// LS Electric XG5000 project: 16-41-1
// PLC NewPLC
// module base 0 slot 0: 입출력 모듈:XBC-DR14E (DC 24V 입력 8점, 릴레이 출력 6점)

PROGRAM NewProgram (task: 스캔 프로그램)

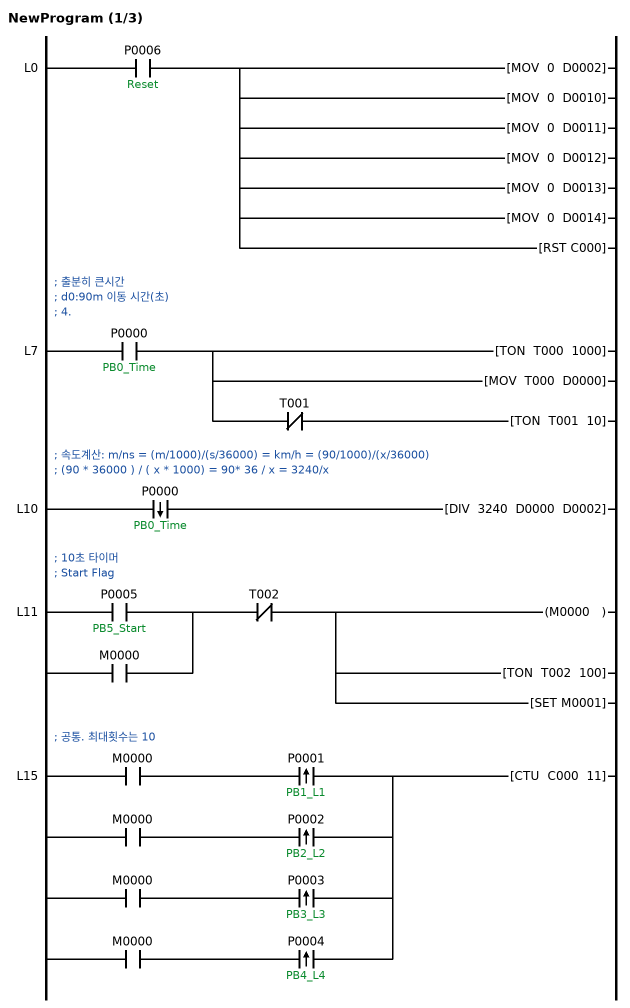
; L0
LOAD      P0006	// Reset
MOV       0 D0002
MOV       0 D0010
MOV       0 D0011
MOV       0 D0012
MOV       0 D0013
MOV       0 D0014
RST       C000
; L7
LOAD      P0000	// PB0_Time
TON       T000 1000
MOV       T000 D0000
AND NOT   T001
TON       T001 10
// output comment: 출분히 큰시간
// output comment: d0:90m 이동 시간(초)
// output comment: 4.
; L10
LOADN     P0000	// PB0_Time
DIV       3240 D0000 D0002
// output comment: 속도계산: m/ns = (m/1000)/(s/36000) = km/h = (90/1000)/(x/36000)           (90 * 36000 ) / ( x * 1000) = 90* 36 / x = 3240/x
; L11
LOAD      P0005	// PB5_Start
OR        M0000
AND NOT   T002
OUT       M0000
TON       T002 100
SET       M0001
// output comment: 10초 타이머
// output comment: Start Flag
; L15
LOAD      M0000
ANDP      P0001	// PB1_L1
LOAD      M0000
ANDP      P0002	// PB2_L2
OR LOAD
LOAD      M0000
ANDP      P0003	// PB3_L3
OR LOAD
LOAD      M0000
ANDP      P0004	// PB4_L4
OR LOAD
CTU       C000 11
// output comment: 공통. 최대횟수는 10

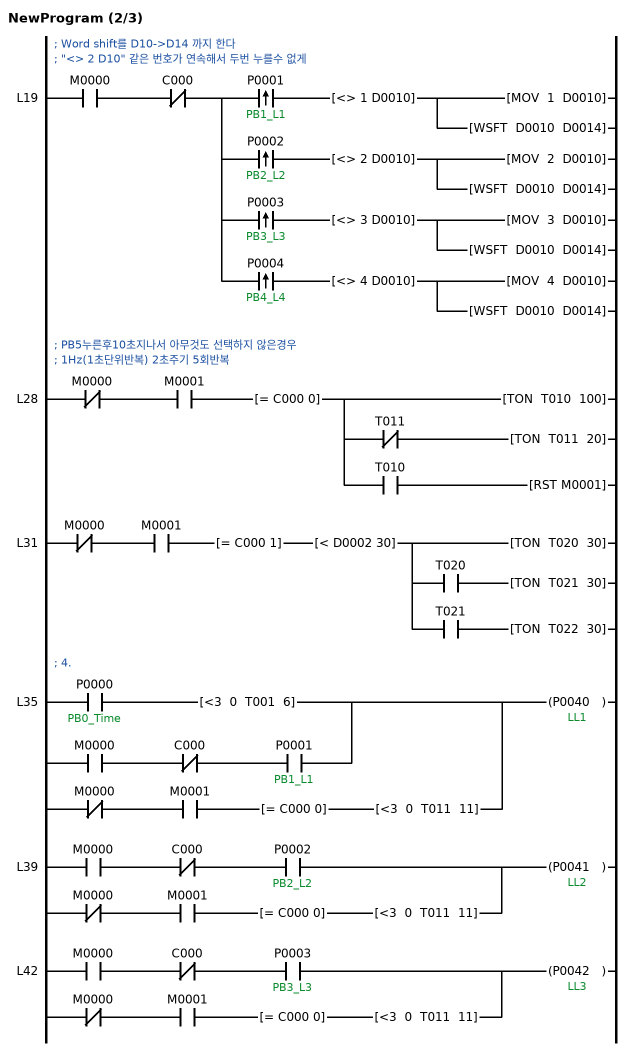
; L19
LOAD      M0000
AND NOT   C000
MPUSH
ANDP      P0001	// PB1_L1
AND<>     1 D0010
MOV       1 D0010
WSFT      D0010 D0014
MLOAD
ANDP      P0002	// PB2_L2
AND<>     2 D0010
MOV       2 D0010
WSFT      D0010 D0014
MLOAD
ANDP      P0003	// PB3_L3
AND<>     3 D0010
MOV       3 D0010
WSFT      D0010 D0014
MPOP
ANDP      P0004	// PB4_L4
AND<>     4 D0010
MOV       4 D0010
WSFT      D0010 D0014
// output comment: Word shift를 D10->D14 까지 한다
// output comment: "<> 2 D10" 같은 번호가 연속해서 두번 누를수 없게 
; L28
LOAD NOT  M0000
AND       M0001
AND=      C000 0
TON       T010 100
MPUSH
AND NOT   T011
TON       T011 20
MPOP
AND       T010
RST       M0001
// output comment: PB5누른후10초지나서 아무것도 선택하지 않은경우
// output comment: 1Hz(1초단위반복) 2초주기 5회반복
; L31
LOAD NOT  M0000
AND       M0001
AND=      C000 1
AND<      D0002 30
TON       T020 30
MPUSH
AND       T020
TON       T021 30
MPOP
AND       T021
TON       T022 30
; L35
LOAD      P0000	// PB0_Time
AND<3     0 T001 6
LOAD      M0000
AND NOT   C000
AND       P0001	// PB1_L1
OR LOAD
LOAD NOT  M0000
AND       M0001
AND=      C000 0
AND<3     0 T011 11
OR LOAD
OUT       P0040	// LL1
// output comment: 4.
; L39
LOAD      M0000
AND NOT   C000
AND       P0002	// PB2_L2
LOAD NOT  M0000
AND       M0001
AND=      C000 0
AND<3     0 T011 11
OR LOAD
OUT       P0041	// LL2
; L42
LOAD      M0000
AND NOT   C000
AND       P0003	// PB3_L3
LOAD NOT  M0000
AND       M0001
AND=      C000 0
AND<3     0 T011 11
OR LOAD
OUT       P0042	// LL3

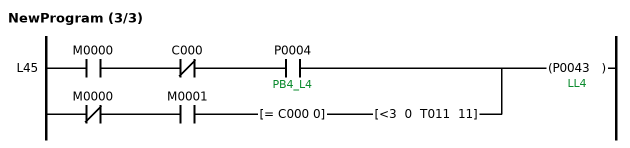
; L45
LOAD      M0000
AND NOT   C000
AND       P0004	// PB4_L4
LOAD NOT  M0000
AND       M0001
AND=      C000 0
AND<3     0 T011 11
OR LOAD
OUT       P0043	// LL4